
// ===== library: MasterCopy "clampDInt" =====

// folder: clamp

FUNCTION "clampDInt" : Void   // FC11, LAD
TITLE = Standard Function CLAMP (DOUBLE INT)
{ S7_Optimized_Access := 'TRUE' }
VERSION : 0.1
// CLAMP function is designed to guarantee the client (user whom call it) that a variable is contained into upper and lower limits.
// If the value is major of max then it is forced to max value.
// If the value is minor of min then it is forced to min value.
   VAR_INPUT
      min : DInt;
      max : DInt;
   END_VAR
   VAR_IN_OUT
      value : DInt;
   END_VAR
BEGIN

REGION Network 1: Maximum value control.
   // execute control and force the value if needed.
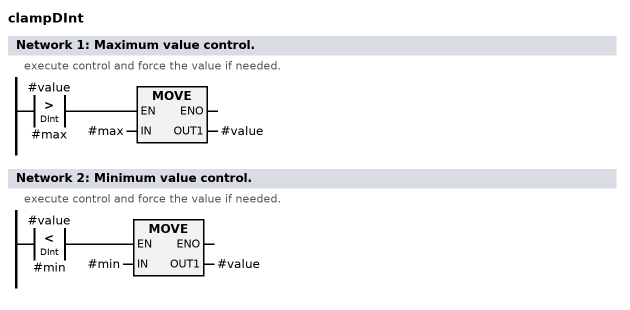
   RUNG wire#powerrail
      { S7_Templates := "SrcType := DInt" } GT_Contact(in1 := #value, in2 := #max)
      Move(in := #max, out1 => #value)
   END_RUNG
   // the same network as SCL:
   IF #value > #max THEN #value := #max; END_IF;
END_REGION

REGION Network 2: Minimum value control.
   // execute control and force the value if needed.
   RUNG wire#powerrail
      { S7_Templates := "SrcType := DInt" } LT_Contact(in1 := #value, in2 := #min)
      Move(in := #min, out1 => #value)
   END_RUNG
   // the same network as SCL:
   IF #value < #min THEN #value := #min; END_IF;
END_REGION
END_FUNCTION

// ===== library: MasterCopy "clampInt" =====

// folder: clamp

FUNCTION "clampInt" : Void   // FC9, LAD
TITLE = Standard Function CLAMP (INTEGERS)
{ S7_Optimized_Access := 'TRUE' }
VERSION : 0.1
// CLAMP function is designed to guarantee the client (user whom call it) that a variable is contained into upper and lower limits.
// If the value is major of max then it is forced to max value.
// If the value is minor of min then it is forced to min value.
   VAR_INPUT
      min : Int;
      max : Int;
   END_VAR
   VAR_IN_OUT
      value : Int;
   END_VAR
BEGIN

REGION Network 1: Maximum value control.
   // execute control and force the value if needed.
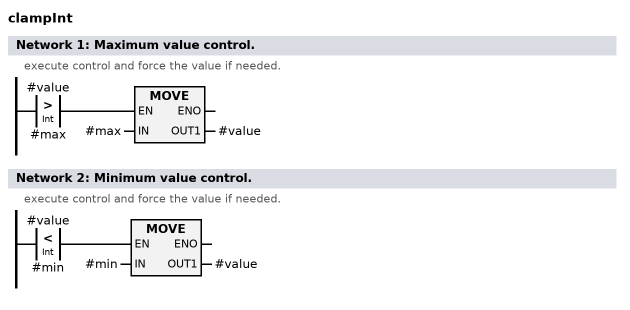
   RUNG wire#powerrail
      { S7_Templates := "SrcType := Int" } GT_Contact(in1 := #value, in2 := #max)
      Move(in := #max, out1 => #value)
   END_RUNG
   // the same network as SCL:
   IF #value > #max THEN #value := #max; END_IF;
END_REGION

REGION Network 2: Minimum value control.
   // execute control and force the value if needed.
   RUNG wire#powerrail
      { S7_Templates := "SrcType := Int" } LT_Contact(in1 := #value, in2 := #min)
      Move(in := #min, out1 => #value)
   END_RUNG
   // the same network as SCL:
   IF #value < #min THEN #value := #min; END_IF;
END_REGION
END_FUNCTION

// ===== library: MasterCopy "clampReal" =====

// folder: clamp

FUNCTION "clampReal" : Void   // FC8, LAD
TITLE = Standard Function CLAMP (REAL)
{ S7_Optimized_Access := 'TRUE' }
VERSION : 0.1
// CLAMP function is designed to guarantee the client (user whom call it) that a variable is contained into upper and lower limits.
// If the value is major of max then it is forced to max value.
// If the value is minor of min then it is forced to min value.
   VAR_INPUT
      min : Real;
      max : Real;
   END_VAR
   VAR_IN_OUT
      value : Real;
   END_VAR
BEGIN

REGION Network 1: Maximum value control.
   // execute control and force the value if needed.
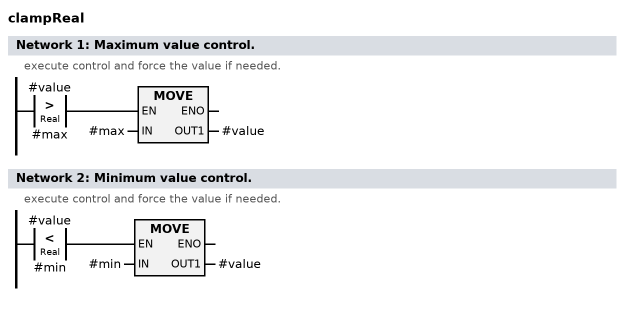
   RUNG wire#powerrail
      { S7_Templates := "SrcType := Real" } GT_Contact(in1 := #value, in2 := #max)
      Move(in := #max, out1 => #value)
   END_RUNG
   // the same network as SCL:
   IF #value > #max THEN #value := #max; END_IF;
END_REGION

REGION Network 2: Minimum value control.
   // execute control and force the value if needed.
   RUNG wire#powerrail
      { S7_Templates := "SrcType := Real" } LT_Contact(in1 := #value, in2 := #min)
      Move(in := #min, out1 => #value)
   END_RUNG
   // the same network as SCL:
   IF #value < #min THEN #value := #min; END_IF;
END_REGION
END_FUNCTION

// ===== library: MasterCopy "PID" =====

FUNCTION_BLOCK "PID"   // FB18, LAD
TITLE = PID (also RAMP if P is off)
{ S7_Optimized_Access := 'FALSE' }
VERSION : 0.1
// PI control. 
// 
// NOTE: D control has to be developed.
// 
// NOTE: It can be used as RAMP while Proportional Action is Off
   VAR_INPUT
      Activate : Bool;
      Freeze : Bool;   // Sospende integrazione
      Reinitialize : Bool;
      OUT_INIT_VAL : Real;   // Posizione asse all'avvio della regolazione
      SP : Real;
      PV : Real;
      OUT_MIN_LIMIT : Real;
      OUT_MAX_LIMIT : Real;
   END_VAR
   VAR_IN_OUT
      OUT_CTRL_VALUE : Real;
   END_VAR
   VAR
      INTEGRAL_COMPONENT : Struct
         I_ON : Bool;   // Attiva componente I nel caso true
         I_SP : Real;   // Coefficiente integrale
         I_DeadBand_SP : Real;
         I_MIN_LIMIT_SP : Real;   // Valore limite integratore MIN
         I_MAX_LIMIT_SP : Real;   // Valore limite integratore MAX
         DEADBAND_HIGH_SP_CALC : Real;   // Sp + deadband
         DEADBAND_LOW_SP_CALC : Real;   // Sp - deadband
         I_INC_LOGIC : Bool;   // logica plc richiede incremento valore act
         I_DEC_LOGIC : Bool;   // logica plc richiede decremento valore act
         ACT_VALUE : Real;   // Valore attuale componente I
      END_STRUCT;
      PROPORTIONAL_COMPONENT : Struct
         P_ON : Bool;
         K_SP : Real;   // Coefficiente proporzionale
         ERR_COMPONENT : Real;
         ERR_COMPONENT_MUL_K : Real;
      END_STRUCT;
      AUX : Struct
         ActivatePulse : Bool;
         auxActivatePulse : Bool;
         initialValueSaved : Real;
      END_STRUCT;
   END_VAR
   VAR_TEMP
      ON : Bool;
      OFF : Bool;
   END_VAR
   VAR_TEMP   // added for the SCL form of the ladder/FBD networks
      _w1 : Bool;
      _w2 : Bool;
   END_VAR
BEGIN

REGION Network 1: Always ON internal flag
   // Always on flag
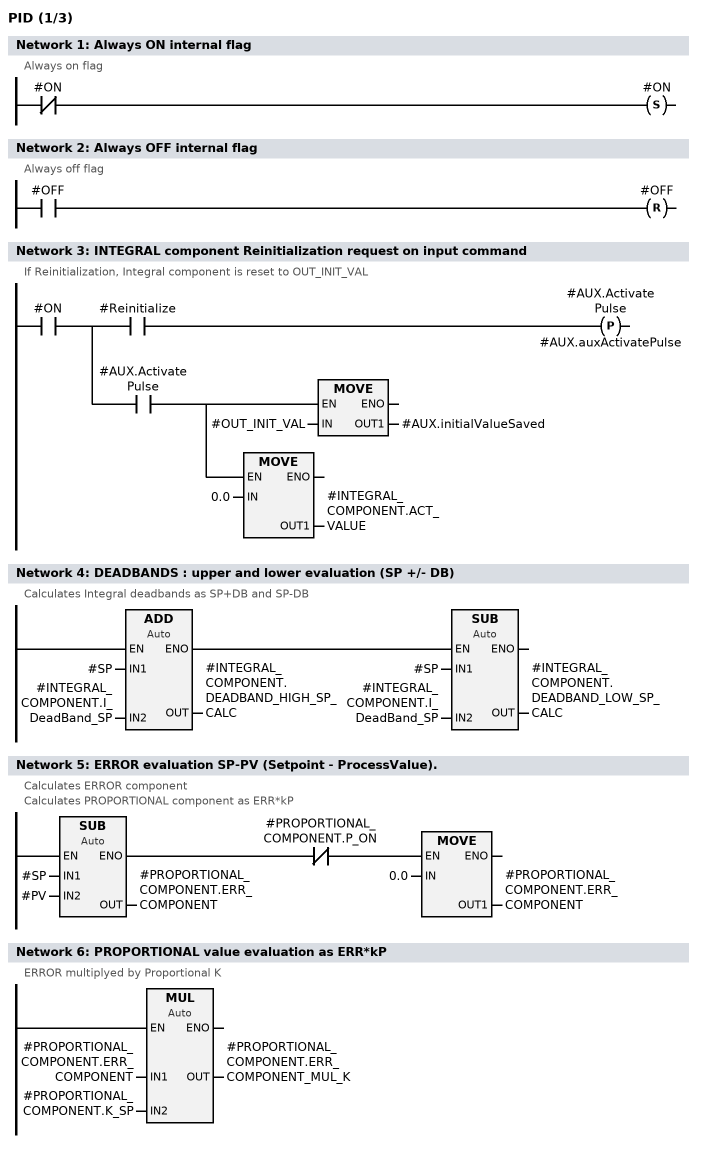
   RUNG wire#powerrail
      I_Contact( #ON )
      S_Coil( #ON )
   END_RUNG
   // the same network as SCL:
   IF NOT #ON THEN #ON := TRUE; END_IF;
END_REGION

REGION Network 2: Always OFF internal flag
   // Always off flag
   RUNG wire#powerrail
      Contact( #OFF )
      R_Coil( #OFF )
   END_RUNG
   // the same network as SCL:
   IF #OFF THEN #OFF := FALSE; END_IF;
END_REGION

REGION Network 3: INTEGRAL component Reinitialization request on input command
   // If Reinitialization, Integral component is reset to OUT_INIT_VAL
   #_w1 := #ON AND #Reinitialize;
   #AUX.ActivatePulse := #_w1 AND NOT #AUX.auxActivatePulse;   // rising edge
   #AUX.auxActivatePulse := #_w1;
   IF #ON AND #AUX.ActivatePulse THEN
       #AUX.initialValueSaved := #OUT_INIT_VAL;
       #INTEGRAL_COMPONENT.ACT_VALUE := 0.0;
   END_IF;
END_REGION

REGION Network 4: DEADBANDS : upper and lower evaluation (SP +/- DB)
   // Calculates Integral deadbands as SP+DB and SP-DB
   RUNG wire#powerrail
      Add(in1 := #SP, in2 := #INTEGRAL_COMPONENT.I_DeadBand_SP, out => #INTEGRAL_COMPONENT.DEADBAND_HIGH_SP_CALC)
      Sub(in1 := #SP, in2 := #INTEGRAL_COMPONENT.I_DeadBand_SP, out => #INTEGRAL_COMPONENT.DEADBAND_LOW_SP_CALC)
   END_RUNG
   // the same network as SCL:
   #INTEGRAL_COMPONENT.DEADBAND_HIGH_SP_CALC := #SP + #INTEGRAL_COMPONENT.I_DeadBand_SP;
   #INTEGRAL_COMPONENT.DEADBAND_LOW_SP_CALC := #SP - #INTEGRAL_COMPONENT.I_DeadBand_SP;
END_REGION

REGION Network 5: ERROR evaluation SP-PV (Setpoint - ProcessValue).
   // Calculates ERROR component
   // Calculates PROPORTIONAL component as ERR*kP
   RUNG wire#powerrail
      Sub(in1 := #SP, in2 := #PV, out => #PROPORTIONAL_COMPONENT.ERR_COMPONENT)
      I_Contact( #PROPORTIONAL_COMPONENT.P_ON )
      Move(in := 0.0, out1 => #PROPORTIONAL_COMPONENT.ERR_COMPONENT)
   END_RUNG
   // the same network as SCL:
   #PROPORTIONAL_COMPONENT.ERR_COMPONENT := #SP - #PV;
   IF NOT #PROPORTIONAL_COMPONENT.P_ON THEN #PROPORTIONAL_COMPONENT.ERR_COMPONENT := 0.0; END_IF;
END_REGION

REGION Network 6: PROPORTIONAL value evaluation as ERR*kP
   // ERROR multiplyed by Proportional K
   RUNG wire#powerrail
      Mul(in1 := #PROPORTIONAL_COMPONENT.ERR_COMPONENT, in2 := #PROPORTIONAL_COMPONENT.K_SP, out => #PROPORTIONAL_COMPONENT.ERR_COMPONENT_MUL_K)
   END_RUNG
   // the same network as SCL:
   #PROPORTIONAL_COMPONENT.ERR_COMPONENT_MUL_K := #PROPORTIONAL_COMPONENT.ERR_COMPONENT * #PROPORTIONAL_COMPONENT.K_SP;
END_REGION

REGION Network 7: INTEGRAL action evaluation(CLAMPED to MIN/MAX)
   // Evaluates if INTEGRAL action has to INCREASE or DECREASE.
   // If limits are surpassed, a clamp action restores consistent values for integral internal variable.
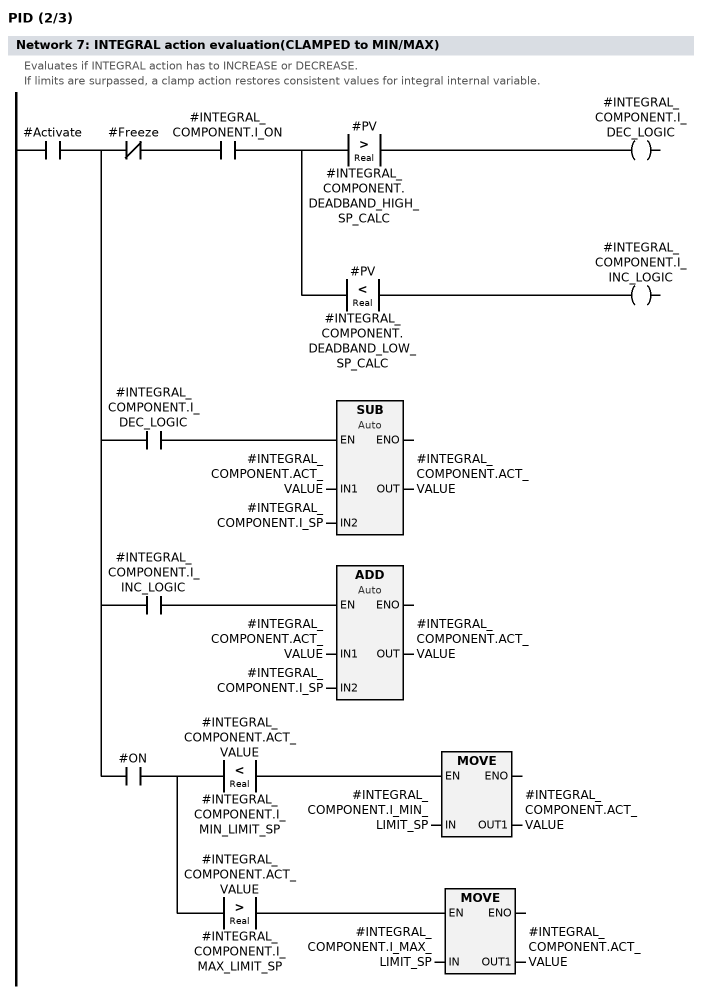
   RUNG wire#powerrail
      Contact( #Activate )
      wire#w1
      I_Contact( #Freeze )
      Contact( #INTEGRAL_COMPONENT.I_ON )
      wire#w2
      { S7_Templates := "SrcType := Real" } GT_Contact(in1 := #PV, in2 := #INTEGRAL_COMPONENT.DEADBAND_HIGH_SP_CALC)
      Coil( #INTEGRAL_COMPONENT.I_DEC_LOGIC )
   END_RUNG
   RUNG wire#w2
      { S7_Templates := "SrcType := Real" } LT_Contact(in1 := #PV, in2 := #INTEGRAL_COMPONENT.DEADBAND_LOW_SP_CALC)
      Coil( #INTEGRAL_COMPONENT.I_INC_LOGIC )
   END_RUNG
   RUNG wire#w1
      Contact( #INTEGRAL_COMPONENT.I_DEC_LOGIC )
      Sub(in1 := #INTEGRAL_COMPONENT.ACT_VALUE, in2 := #INTEGRAL_COMPONENT.I_SP, out => #INTEGRAL_COMPONENT.ACT_VALUE)
   END_RUNG
   RUNG wire#w1
      Contact( #INTEGRAL_COMPONENT.I_INC_LOGIC )
      Add(in1 := #INTEGRAL_COMPONENT.ACT_VALUE, in2 := #INTEGRAL_COMPONENT.I_SP, out => #INTEGRAL_COMPONENT.ACT_VALUE)
   END_RUNG
   RUNG wire#w1
      Contact( #ON )
      wire#w3
      { S7_Templates := "SrcType := Real" } LT_Contact(in1 := #INTEGRAL_COMPONENT.ACT_VALUE, in2 := #INTEGRAL_COMPONENT.I_MIN_LIMIT_SP)
      Move(in := #INTEGRAL_COMPONENT.I_MIN_LIMIT_SP, out1 => #INTEGRAL_COMPONENT.ACT_VALUE)
   END_RUNG
   RUNG wire#w3
      { S7_Templates := "SrcType := Real" } GT_Contact(in1 := #INTEGRAL_COMPONENT.ACT_VALUE, in2 := #INTEGRAL_COMPONENT.I_MAX_LIMIT_SP)
      Move(in := #INTEGRAL_COMPONENT.I_MAX_LIMIT_SP, out1 => #INTEGRAL_COMPONENT.ACT_VALUE)
   END_RUNG
   // the same network as SCL:
   #_w1 := #Activate AND NOT #Freeze AND #INTEGRAL_COMPONENT.I_ON;
   #INTEGRAL_COMPONENT.I_DEC_LOGIC := #_w1 AND (#PV > #INTEGRAL_COMPONENT.DEADBAND_HIGH_SP_CALC);
   #INTEGRAL_COMPONENT.I_INC_LOGIC := #_w1 AND (#PV < #INTEGRAL_COMPONENT.DEADBAND_LOW_SP_CALC);
   IF #Activate AND #INTEGRAL_COMPONENT.I_DEC_LOGIC THEN
       #INTEGRAL_COMPONENT.ACT_VALUE := #INTEGRAL_COMPONENT.ACT_VALUE - #INTEGRAL_COMPONENT.I_SP;
   END_IF;
   IF #Activate AND #INTEGRAL_COMPONENT.I_INC_LOGIC THEN
       #INTEGRAL_COMPONENT.ACT_VALUE := #INTEGRAL_COMPONENT.ACT_VALUE + #INTEGRAL_COMPONENT.I_SP;
   END_IF;
   #_w2 := #Activate AND #ON;
   IF #_w2 AND (#INTEGRAL_COMPONENT.ACT_VALUE < #INTEGRAL_COMPONENT.I_MIN_LIMIT_SP) THEN
       #INTEGRAL_COMPONENT.ACT_VALUE := #INTEGRAL_COMPONENT.I_MIN_LIMIT_SP;
   END_IF;
   IF #_w2 AND (#INTEGRAL_COMPONENT.ACT_VALUE > #INTEGRAL_COMPONENT.I_MAX_LIMIT_SP) THEN
       #INTEGRAL_COMPONENT.ACT_VALUE := #INTEGRAL_COMPONENT.I_MAX_LIMIT_SP;
   END_IF;
END_REGION

REGION Network 8: OUTPUT control value evaluation as P+I
   // Add P component and I component
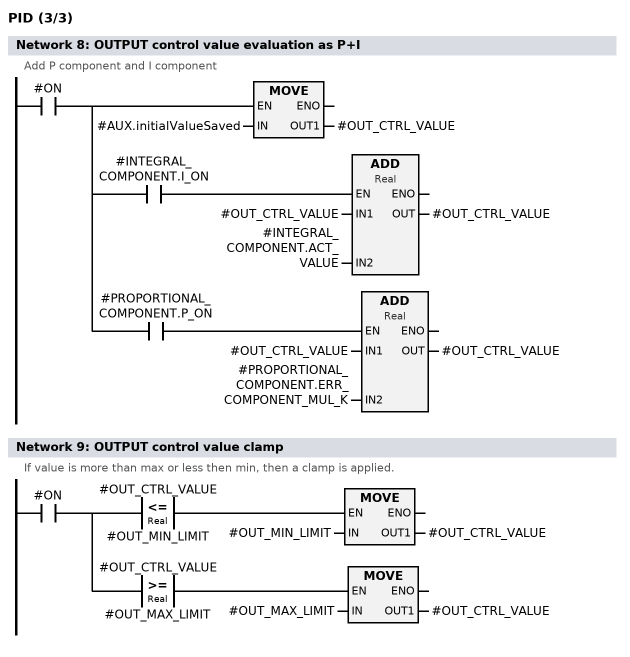
   RUNG wire#powerrail
      Contact( #ON )
      wire#w1
      Move(in := #AUX.initialValueSaved, out1 => #OUT_CTRL_VALUE)
   END_RUNG
   RUNG wire#w1
      Contact( #INTEGRAL_COMPONENT.I_ON )
      { S7_Templates := "SrcType := Real" } Add(in1 := #OUT_CTRL_VALUE, in2 := #INTEGRAL_COMPONENT.ACT_VALUE, out => #OUT_CTRL_VALUE)
   END_RUNG
   RUNG wire#w1
      Contact( #PROPORTIONAL_COMPONENT.P_ON )
      { S7_Templates := "SrcType := Real" } Add(in1 := #OUT_CTRL_VALUE, in2 := #PROPORTIONAL_COMPONENT.ERR_COMPONENT_MUL_K, out => #OUT_CTRL_VALUE)
   END_RUNG
   // the same network as SCL:
   IF #ON THEN #OUT_CTRL_VALUE := #AUX.initialValueSaved; END_IF;
   IF #ON AND #INTEGRAL_COMPONENT.I_ON THEN
       #OUT_CTRL_VALUE := #OUT_CTRL_VALUE + #INTEGRAL_COMPONENT.ACT_VALUE;
   END_IF;
   IF #ON AND #PROPORTIONAL_COMPONENT.P_ON THEN
       #OUT_CTRL_VALUE := #OUT_CTRL_VALUE + #PROPORTIONAL_COMPONENT.ERR_COMPONENT_MUL_K;
   END_IF;
END_REGION

REGION Network 9: OUTPUT control value clamp
   // If value is more than max or less then min, then a clamp is applied.
   RUNG wire#powerrail
      Contact( #ON )
      wire#w1
      { S7_Templates := "SrcType := Real" } LE_Contact(in1 := #OUT_CTRL_VALUE, in2 := #OUT_MIN_LIMIT)
      Move(in := #OUT_MIN_LIMIT, out1 => #OUT_CTRL_VALUE)
   END_RUNG
   RUNG wire#w1
      { S7_Templates := "SrcType := Real" } GE_Contact(in1 := #OUT_CTRL_VALUE, in2 := #OUT_MAX_LIMIT)
      Move(in := #OUT_MAX_LIMIT, out1 => #OUT_CTRL_VALUE)
   END_RUNG
   // the same network as SCL:
   IF #ON AND (#OUT_CTRL_VALUE <= #OUT_MIN_LIMIT) THEN #OUT_CTRL_VALUE := #OUT_MIN_LIMIT; END_IF;
   IF #ON AND (#OUT_CTRL_VALUE >= #OUT_MAX_LIMIT) THEN #OUT_CTRL_VALUE := #OUT_MAX_LIMIT; END_IF;
END_REGION
END_FUNCTION_BLOCK

// ===== library: MasterCopy "linearReal" =====

FUNCTION "linearReal" : Void   // FC17, SCL
{ S7_Optimized_Access := 'TRUE' }
VERSION : 0.1
   VAR_INPUT
      Value : Real;
      ValueMin : Real;
      ValueMax : Real;
      OutMin : Real;
      OutMax : Real;
   END_VAR
   VAR_OUTPUT
      OUTPUT : Real;
      ERR : Bool;
   END_VAR
   VAR_TEMP
      DeltaIn : Real;
      DeltaOut : Real;
      Kappa : Real;
      ValueShift : Real;
   END_VAR
BEGIN
   // Verifica input in range o fuori range
   IF #Value < #ValueMin OR #Value > #ValueMax THEN
       #ERR := true;
   ELSE
       #ERR := false;

       #DeltaIn := #ValueMax - #ValueMin;
       #DeltaOut := #OutMax - #OutMin;
       #Kappa := #DeltaOut / #DeltaIn;
       #ValueShift := #Value - #ValueMin;
       #OUTPUT := (#ValueShift * #Kappa) + #OutMin;
   END_IF;
END_FUNCTION